FUNCTION_BLOCK "Semantic_ReferenceManualInitializer"
{ S7_Optimized_Access := 'TRUE' }
VERSION : 0.1

VAR_TEMP
    badReference : REF_TO Int := NULL;
    // EXPECT: error[reference.manual-initial-value-forbidden] SEM-REF-005
END_VAR

BEGIN
END_FUNCTION_BLOCK
